// Mitsubishi GX Works2 project: Stepper1   PLC: FX2N/FX2NC

PROGRAM MAIN
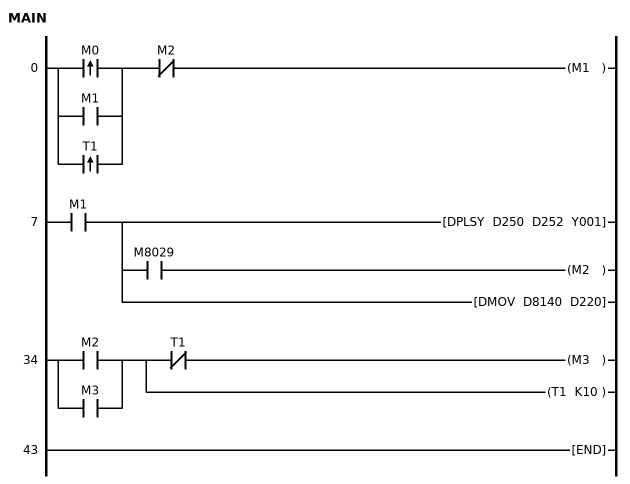
0     LDP     M0
      OR      M1
      ORP     T1
      ANI     M2
      OUT     M1
7     LD      M1
      DPLSY   D250 D252 Y001
      MPS
      AND     M8029
      OUT     M2
      MPP
      DMOV    D8140 D220
34    LD      M2
      OR      M3
      MPS
      ANI     T1
      OUT     M3
      MPP
      OUT     T1 K10
43    END
END_PROGRAM
